// TIA Portal V16 export
// export: Created 2024-12-03T15:41:41.7978577Z, ExportSetting WithDefaults, DisplayName Totally Integrated Automation Portal, DisplayVersion V16 Update 6, DisplayName TIA Portal Version Control Interface, DisplayVersion V16 Update 2, DisplayName TIA Portal Openness, DisplayVersion V16 Update 6, DisplayName TIA Portal Teamcenter Gateway, DisplayVersion V16, DisplayName SINAMICS Startdrive Advanced, DisplayVersion V16 Update 5, DisplayName SINAMICS Startdrive G130, G150, S120, S150, SINAMICS MV, S210, DisplayVersion V16 Update 5, DisplayName SINAMICS Startdrive G110M, G120, G120C, G120D, G120P, G115D, DisplayVersion V16 Update 5, DisplayName STEP 7 Professional, DisplayVersion V16 Update 6, DisplayName STEP 7 Safety, DisplayVersion V16, DisplayName WinCC Advanced / Unified PC, DisplayVersion V16 Update 6
FUNCTION_BLOCK "EasySystems_TransferUnit_UpDown_Controller_FB"   // FB33, SCL
{ S7_Optimized_Access := 'TRUE' }
VERSION : 0.1
// stored: AutoNumber true, IsIECCheckEnabled false, IsRetainMemResEnabled false, MemoryReserve 100, SetENOAutomatically false, UDAEnableTagReadback false
   VAR_INPUT
      I_MotorData : "CLXAiPLC_IN_UDT";   // The 64 byte input word of the IO module
      I_ControlLeftMotorConveyLInx : Bool;   // 1 = control left motor both motos can be controlled with one module
      I_ControlRightMotorConveyLinx : Bool;   // 1 = control right motor both motors can be controlled with one fb
      I_UpFb : Bool;   // Object is up feedback
      I_DownFb : Bool;   // Object is down feedback
      I_TimeUp : Time := t#5s;   // time to go up
      I_TimeDown : Time := t#5s;   // time to go down
      I_Direction : Bool;   // Direction of the motor
   END_VAR
   VAR_IN_OUT
      IO_MotorStatus : "EasySystems_LineairMotor_ConveyLinx_FullPLC_Single";
      IO_MotorOutput : "CLXAiPLC_OUT_UDT";   // All the motor commands
   END_VAR
   VAR
      SensorUp : "SmartBool";
      SensorDown : "SmartBool";
      NotConnected { S7_SetPoint := 'True'} : TON_TIME;
      NotUp { S7_SetPoint := 'True'} : TON_TIME;
      NotDown { S7_SetPoint := 'True'} : TON_TIME;
      srUp { S7_SetPoint := 'True'} : "SR";
      srDown { S7_SetPoint := 'True'} : "SR";
      CycleRun { S7_SetPoint := 'True'} : "CycleRun";
   END_VAR
   VAR DB_SPECIFIC
      AlarmInfo { S7_SetPoint := 'True'} : "AlarmInfo_UDT";
   END_VAR
   VAR
      Overheat { S7_SetPoint := 'True'} : Program_Alarm;
      ShortCircuit { S7_SetPoint := 'True'} : Program_Alarm;
      MDRNotConnected { S7_SetPoint := 'True'} : Program_Alarm;
      Overload { S7_SetPoint := 'True'} : Program_Alarm;
      Stalled { S7_SetPoint := 'True'} : Program_Alarm;
      MDRBadHall { S7_SetPoint := 'True'} : Program_Alarm;
      OverVoltage { S7_SetPoint := 'True'} : Program_Alarm;
      LowVoltage { S7_SetPoint := 'True'} : Program_Alarm;
      NotConnectedAlarm { S7_SetPoint := 'True'} : Program_Alarm;
      ConnectionNotOK { S7_SetPoint := 'True'} : Program_Alarm;
      AnyErrorActive { S7_SetPoint := 'True'} : Program_Alarm;
      JamError { S7_SetPoint := 'True'} : Program_Alarm;
      SensorLowGain { S7_SetPoint := 'True'} : Program_Alarm;
      NotUpAlarm { S7_SetPoint := 'True'} : Program_Alarm;
      NotDownAlarm { S7_SetPoint := 'True'} : Program_Alarm;
   END_VAR
   VAR_TEMP
      T_RunAuto : Bool;
      T_RunManual : Bool;
      T_AppState : "ApplicationState_UDT";
      T_ZoneInfo : "ZoneInfo";
   END_VAR
BEGIN
   #T_ZoneInfo := "ApplicationState_DB".ZoneNames[#IO_MotorStatus.Zone];
   #T_AppState := "ApplicationState_DB".Appstate[#T_ZoneInfo.AppStateIndex];
   #CycleRun(I_End:=15);

   REGION SENSOR INTERFACING

       #SensorUp(I_Sensor:=#I_UpFb);
       #SensorDown(I_Sensor := #I_DownFb);

   END_REGION

   REGION Commands

       //Transfer unit settings
       #IO_MotorStatus.Cmd.Accel := 80;
       #IO_MotorStatus.Cmd.Deaccel := 1;
       #IO_MotorStatus.Cmd.SpeedManual := 20;
       #IO_MotorStatus.Cmd.SpeedAuto := 20;
       #IO_MotorStatus.Cmd.BrakeMode := 16#3;

       #IO_MotorStatus.Status.ManualCommandsDisabled := 0;

       //Reset commands left
       IF #I_ControlLeftMotorConveyLInx THEN
           #IO_MotorOutput.LeftMDRControl.MDR_Direction := 0;
           #IO_MotorOutput.LeftMDRControl.Run_MDR := 0;
           #IO_MotorOutput.LeftMDRSpeed := 0;
           #IO_MotorOutput.ServoControlCommandLeft.ResetPulseCount := 0;
           #IO_MotorOutput.ServoControlCommandLeft.RunToSetpoint := 0;
           #IO_MotorOutput.LeftMDRAccel := #IO_MotorStatus.Cmd.Accel;
           #IO_MotorOutput.LeftMDRDeccel := #IO_MotorStatus.Cmd.Deaccel;
           #IO_MotorOutput.LeftMDRBrakeMode := #IO_MotorStatus.Cmd.BrakeMode;
       END_IF;

       //Reset commands right
       IF #I_ControlRightMotorConveyLinx THEN
           #IO_MotorOutput.RightMDRControl.MDR_Direction := 0;
           #IO_MotorOutput.RightMDRControl.Run_MDR := 0;
           #IO_MotorOutput.RightMDRSpeed := 0;
           #IO_MotorOutput.ServoControlCommandRight.ResetPulseCount := 0;
           #IO_MotorOutput.ServoControlCommandRight.RunToSetpoint := 0;
           #IO_MotorOutput.RightMDRAccel := #IO_MotorStatus.Cmd.Accel;
           #IO_MotorOutput.RightMDRDeccel := #IO_MotorStatus.Cmd.Deaccel;
           #IO_MotorOutput.RightMDRBrakeMode := #IO_MotorStatus.Cmd.BrakeMode;
       END_IF;

       //INIT command
       IF #IO_MotorStatus.Cmd.InitPosition THEN
           #IO_MotorStatus.Status.PositionLineair := 0;
           #IO_MotorStatus.Cmd.InitPosition := FALSE;
       END_IF;

       IF #IO_MotorStatus.Status.PositionLineair = 1 THEN
           #IO_MotorStatus.Cmd.UpManual := 0;
           #IO_MotorStatus.Cmd.UpAuto := 0;
       END_IF;

       IF #IO_MotorStatus.Status.PositionLineair = -1 THEN
           #IO_MotorStatus.Cmd.DownAuto := 0;
           #IO_MotorStatus.Cmd.DownManual := 0;
       END_IF;

       IF #SensorUp.O_data.LE OR #SensorDown.O_data.LE THEN
           #IO_MotorStatus.Status.ManualCommandsDisabled := 1;
       END_IF;

       #T_RunAuto := #IO_MotorStatus.Cmd.UpAuto OR #IO_MotorStatus.Cmd.DownAuto;
       #T_RunManual := #IO_MotorStatus.Cmd.UpManual OR #IO_MotorStatus.Cmd.DownManual;

       //Turn commands of if manual mode is deactivated
       IF NOT #T_AppState.States.ManualModeActivated.State THEN
           #IO_MotorStatus.Cmd.UpManual := 0;
           #IO_MotorStatus.Cmd.DownManual := 0;
           #T_RunManual := 0;
           #IO_MotorStatus.Status.ManualCommandsDisabled := 1;
       END_IF;

       //Turn commands of if auto mode is deactivated
       IF NOT #T_AppState.States.AutoModeActivated.State THEN
           #IO_MotorStatus.Cmd.UpAuto := 0;
           #IO_MotorStatus.Cmd.DownAuto := 0;
           #T_RunAuto := 0;
       END_IF;

       //Turn commands of if interlock or alarm
       IF #IO_MotorStatus.Alarms.Status > 0 OR #IO_MotorStatus.Alarms.MdrAlarms.Status_1 > 0 OR #IO_MotorStatus.Status.Interlocked THEN
           #T_RunAuto := 0;
           #T_RunManual := 0;
           #IO_MotorStatus.Cmd.DownAuto := 0;
           #IO_MotorStatus.Cmd.DownManual := 0;
           #IO_MotorStatus.Cmd.UpAuto := 0;
           #IO_MotorStatus.Cmd.UpManual := 0;
           #IO_MotorStatus.Status.ManualCommandsDisabled := 1;
       END_IF;

       //Auto mode left
       IF #T_AppState.States.AutoModeActivated.State AND #I_ControlLeftMotorConveyLInx THEN
           #IO_MotorOutput.LeftMDRControl.Run_MDR := #T_RunAuto;
           #IO_MotorOutput.LeftMDRControl.MDR_Direction := #I_Direction;
           #IO_MotorOutput.LeftMDRAccel := #IO_MotorStatus.Cmd.Accel;
           #IO_MotorOutput.LeftMDRDeccel := #IO_MotorStatus.Cmd.Deaccel;
           #IO_MotorOutput.LeftMDRSpeed := #IO_MotorStatus.Cmd.SpeedAuto;
           #IO_MotorOutput.LeftMDRBrakeMode := #IO_MotorStatus.Cmd.BrakeMode;
           #IO_MotorOutput.ServoControlCommandLeft.ResetPulseCount := #IO_MotorStatus.Cmd.ServoResetPulseCount;
           #IO_MotorOutput.ServoControlCommandLeft.RunToSetpoint := #IO_MotorStatus.Cmd.ServoRunToSetpoint;
           #IO_MotorOutput.ServoControlDistanceLeft := #IO_MotorStatus.Cmd.ServoControlDistance;
       END_IF;

       //Auto mode right
       IF #T_AppState.States.AutoModeActivated.State AND #I_ControlRightMotorConveyLinx THEN
           #IO_MotorOutput.RightMDRControl.Run_MDR := #T_RunAuto;
           #IO_MotorOutput.RightMDRControl.MDR_Direction := #I_Direction;
           #IO_MotorOutput.RightMDRAccel := #IO_MotorStatus.Cmd.Accel;
           #IO_MotorOutput.RightMDRDeccel := #IO_MotorStatus.Cmd.Deaccel;
           #IO_MotorOutput.RightMDRSpeed := #IO_MotorStatus.Cmd.SpeedAuto;
           #IO_MotorOutput.RightMDRBrakeMode := #IO_MotorStatus.Cmd.BrakeMode;
           #IO_MotorOutput.ServoControlCommandRight.ResetPulseCount := #IO_MotorStatus.Cmd.ServoResetPulseCount;
           #IO_MotorOutput.ServoControlCommandRight.RunToSetpoint := #IO_MotorStatus.Cmd.ServoRunToSetpoint;
           #IO_MotorOutput.ServoControlDistanceRight := #IO_MotorStatus.Cmd.ServoControlDistance;
       END_IF;

       //Manual mode left
       IF #T_AppState.States.ManualModeActivated.State AND #I_ControlLeftMotorConveyLInx THEN
           #IO_MotorOutput.LeftMDRControl.MDR_Direction := #I_Direction;
           #IO_MotorOutput.LeftMDRControl.Run_MDR := #T_RunManual;
           #IO_MotorOutput.LeftMDRSpeed := #IO_MotorStatus.Cmd.SpeedManual;
       END_IF;

       //Manual mode right
       IF #T_AppState.States.ManualModeActivated.State AND #I_ControlRightMotorConveyLinx THEN
           #IO_MotorOutput.RightMDRControl.MDR_Direction := #I_Direction;
           #IO_MotorOutput.RightMDRControl.Run_MDR := #T_RunManual;
           #IO_MotorOutput.RightMDRSpeed := #IO_MotorStatus.Cmd.SpeedManual;
       END_IF;

       //Default commands
       IF  #I_ControlLeftMotorConveyLInx THEN
           #IO_MotorOutput.LeftMDRAccel := #IO_MotorStatus.Cmd.Accel := 30;
           #IO_MotorOutput.LeftMDRDeccel := #IO_MotorStatus.Cmd.Deaccel := 1;
           #IO_MotorOutput.LeftMDRSpeed := #IO_MotorStatus.Cmd.SpeedAuto := 50;
           #IO_MotorOutput.LeftMDRBrakeMode := #IO_MotorStatus.Cmd.BrakeMode;
       END_IF;

       IF #I_ControlRightMotorConveyLinx THEN
           #IO_MotorOutput.RightMDRAccel := #IO_MotorStatus.Cmd.Accel;
           #IO_MotorOutput.RightMDRDeccel := #IO_MotorStatus.Cmd.Deaccel;
           #IO_MotorOutput.RightMDRSpeed := #IO_MotorStatus.Cmd.SpeedAuto;
           #IO_MotorOutput.RightMDRBrakeMode := #IO_MotorStatus.Cmd.BrakeMode;
       END_IF;

   END_REGION

   REGION Interlock motor

       #IO_MotorStatus.Status.Interlocked := #IO_MotorStatus.Cmd.Interlock OR NOT #T_AppState.States.EmergencyOk.State;
       #IO_MotorStatus.Status.Status.%X0 := #IO_MotorStatus.Status.Interlocked;

   END_REGION

   REGION Create status

       //Lineair position
       IF #SensorUp.O_data.State AND NOT #SensorDown.O_data.State THEN
           #IO_MotorStatus.Status.PositionLineair := 1;
       END_IF;

       IF NOT #SensorUp.O_data.State AND #SensorDown.O_data.State THEN
           #IO_MotorStatus.Status.PositionLineair := -1;
       END_IF;

       IF NOT #T_AppState.States.AutoModeActivated.State
           AND NOT #T_AppState.States.ManualModeActivated.State THEN
           #IO_MotorStatus.Status.PositionLineair := 0;
       END_IF;

       REGION simulation

           IF "Simulation_DB".Simulation_On THEN
               IF #IO_MotorStatus.Cmd.UpAuto OR #IO_MotorStatus.Cmd.UpManual THEN
                   #IO_MotorStatus.Status.PositionLineair := "Up";
               END_IF;
           END_IF;

           IF "Simulation_DB".Simulation_On THEN
               IF #IO_MotorStatus.Cmd.DownAuto OR #IO_MotorStatus.Cmd.DownManual THEN
                   #IO_MotorStatus.Status.PositionLineair := "Down";
               END_IF;
           END_IF;

       END_REGION

       //Left
       IF #I_ControlLeftMotorConveyLInx THEN
           #IO_MotorStatus.Status.ActualSpeed := #I_MotorData.LeftMDRRealSpeed;
           #IO_MotorStatus.Status.Current := #I_MotorData.LeftCurrent;
           #IO_MotorStatus.Status.Frequency := #I_MotorData.LeftFreq;
           #IO_MotorStatus.Status.ManualModeActive := #IO_MotorStatus.Cmd.UpManual OR #IO_MotorStatus.Cmd.DownManual;
           #IO_MotorStatus.Status.Position := #I_MotorData.DistanceLeft;
           #IO_MotorStatus.Status.Running := #I_MotorData.LeftMDRRealSpeed > 0 AND #IO_MotorOutput.LeftMDRControl.Run_MDR;
           #IO_MotorStatus.Status.ServoStatus.LastServoCommandExecuted := #I_MotorData.ServoStatusLeft.LastServoCommandExecuted;
           #IO_MotorStatus.Status.ServoStatus.ResetPulseCount_Echo := #I_MotorData.ServoStatusLeft.ResetPulseCount_Echo;
           #IO_MotorStatus.Status.ServoStatus.RunCommand_Echo := #I_MotorData.ServoStatusLeft.RunCommand_Echo;
           #IO_MotorStatus.Status.TemperatureModule := #I_MotorData.ModuleTemp;
           #IO_MotorStatus.Status.TeperatureMDR := #I_MotorData.LeftCalcTemp;
       END_IF;

       //right
       IF #I_ControlRightMotorConveyLinx THEN
           #IO_MotorStatus.Status.ActualSpeed := #I_MotorData.RightMDRRealSpeed;
           #IO_MotorStatus.Status.Current := #I_MotorData.RightCurrent;
           #IO_MotorStatus.Status.Frequency := #I_MotorData.RightFreq;
           #IO_MotorStatus.Status.ManualModeActive := #IO_MotorStatus.Cmd.UpManual OR #IO_MotorStatus.Cmd.DownManual;
           #IO_MotorStatus.Status.Position := #I_MotorData.DistanceRight;
           #IO_MotorStatus.Status.Running := #I_MotorData.RightMDRRealSpeed > 0 AND #IO_MotorOutput.RightMDRControl.Run_MDR;
           #IO_MotorStatus.Status.ServoStatus.LastServoCommandExecuted := #I_MotorData.ServoStatusRight.LastServoCommandExecuted;
           #IO_MotorStatus.Status.ServoStatus.ResetPulseCount_Echo := #I_MotorData.ServoStatusRight.ResetPulseCount_Echo;
           #IO_MotorStatus.Status.ServoStatus.RunCommand_Echo := #I_MotorData.ServoStatusRight.RunCommand_Echo;
           #IO_MotorStatus.Status.TemperatureModule := #I_MotorData.ModuleTemp;
           #IO_MotorStatus.Status.TeperatureMDR := #I_MotorData.RightCalcTemp;
       END_IF;

       REGION Min max voltage

           #IO_MotorStatus.Status.Voltage := #I_MotorData.Voltage;
           IF #I_MotorData.Voltage < #IO_MotorStatus.Status.MinVoltage THEN
               #IO_MotorStatus.Status.MinVoltage := #I_MotorData.Voltage;
           END_IF;

           IF #I_MotorData.Voltage > #IO_MotorStatus.Status.MaxVoltage THEN
               #IO_MotorStatus.Status.MaxVoltage := #I_MotorData.Voltage;
           END_IF;

       END_REGION

       #IO_MotorStatus.Status.ManualModeActive := #T_AppState.States.ManualModeActivated.State;
       #IO_MotorStatus.Status.Status.%X1 := #IO_MotorStatus.Status.Running;
       #IO_MotorStatus.Status.Status.%X2 := #IO_MotorStatus.Status.ManualModeActive;

   END_REGION

   REGION Check alarm active

       IF #I_ControlLeftMotorConveyLInx THEN

           IF #I_MotorData.LeftMDRDiagnostic.LowVoltage THEN
               #IO_MotorStatus.Alarms.MdrAlarms.LowVoltage.Active := True;
           END_IF;

           IF #I_MotorData.LeftMDRDiagnostic.MDRBadHall THEN
               #IO_MotorStatus.Alarms.MdrAlarms.MDRBadHall.Active := True;
           END_IF;

           IF #I_MotorData.LeftMDRDiagnostic.MDRNotConnected THEN
               #IO_MotorStatus.Alarms.MdrAlarms.MDRNotConnected.Active := True;
           END_IF;

           IF #I_MotorData.LeftMDRDiagnostic.Overheat THEN
               #IO_MotorStatus.Alarms.MdrAlarms.Overheat.Active := True;
           END_IF;

           IF #I_MotorData.LeftMDRDiagnostic.Overload THEN
               #IO_MotorStatus.Alarms.MdrAlarms.Overload.Active := True;
           END_IF;

           IF #I_MotorData.LeftMDRDiagnostic.OverVoltage THEN
               #IO_MotorStatus.Alarms.MdrAlarms.OverVoltage.Active := True;
           END_IF;

           IF #I_MotorData.LeftMDRDiagnostic.ShortCircuit THEN
               #IO_MotorStatus.Alarms.MdrAlarms.ShortCircuit.Active := True;
           END_IF;

           IF #I_MotorData.LeftMDRDiagnostic.Stalled THEN
               #IO_MotorStatus.Alarms.MdrAlarms.Stalled.Active := True;
           END_IF;

       END_IF;

       IF #I_ControlRightMotorConveyLinx THEN

           IF #I_MotorData.RightMDRDiagnostic.LowVoltage THEN
               #IO_MotorStatus.Alarms.MdrAlarms.LowVoltage.Active := True;
           END_IF;

           IF #I_MotorData.RightMDRDiagnostic.MDRBadHall THEN
               #IO_MotorStatus.Alarms.MdrAlarms.MDRBadHall.Active := True;
           END_IF;

           IF #I_MotorData.RightMDRDiagnostic.MDRNotConnected THEN
               #IO_MotorStatus.Alarms.MdrAlarms.MDRNotConnected.Active := True;
           END_IF;

           IF #I_MotorData.RightMDRDiagnostic.Overheat THEN
               #IO_MotorStatus.Alarms.MdrAlarms.Overheat.Active := True;
           END_IF;

           IF #I_MotorData.RightMDRDiagnostic.Overload THEN
               #IO_MotorStatus.Alarms.MdrAlarms.Overload.Active := True;
           END_IF;

           IF #I_MotorData.RightMDRDiagnostic.OverVoltage THEN
               #IO_MotorStatus.Alarms.MdrAlarms.OverVoltage.Active := True;
           END_IF;

           IF #I_MotorData.RightMDRDiagnostic.ShortCircuit THEN
               #IO_MotorStatus.Alarms.MdrAlarms.ShortCircuit.Active := True;
           END_IF;

           IF #I_MotorData.RightMDRDiagnostic.Stalled THEN
               #IO_MotorStatus.Alarms.MdrAlarms.Stalled.Active := True;
           END_IF;

       END_IF;

       #IO_MotorStatus.Heartbeat := #I_MotorData.AllSensors.Heartbeat;
       #NotConnected(IN := NOT #IO_MotorStatus.Heartbeat,
                       PT := t#5s);

       IF #NotConnected.Q THEN
           #IO_MotorStatus.Alarms.MdrAlarms.NotConnected.Active := true;
       END_IF;

       //Not up
       #NotUp(IN := (#IO_MotorStatus.Cmd.UpAuto OR #IO_MotorStatus.Cmd.UpManual) AND NOT #SensorUp.O_data.State,
                PT := #I_TimeUp);

       #srUp(I_set := #NotUp.Q,
               I_Reset := #T_AppState.Hmi_Buttons.reset.state.State,
               O_state => #IO_MotorStatus.Alarms.NotUp.Active);

       //Not down
         #NotDown(IN := (#IO_MotorStatus.Cmd.DownAuto OR #IO_MotorStatus.Cmd.DownManual) AND NOT #SensorDown.O_data.State,
                  PT := #I_TimeDown);

       #srDown(I_set := #NotDown.Q,
                 I_Reset := #T_AppState.Hmi_Buttons.reset.state.State,
                 O_state => #IO_MotorStatus.Alarms.NotDown.Active);

       REGION PROGRAM ALARMS

           REGION alarm info
               IF NOT #AlarmInfo.init THEN
                   #IO_MotorStatus.Info.Name := "buildObjectName"(I_Symbolname := GetSymbolName(variable := #IO_MotorStatus,size := 100));
                   #AlarmInfo.info := "buildAlarmInfo"(I_ZoneIndex := #IO_MotorStatus.Zone, I_ZoneName := #T_ZoneInfo.ZoneName, I_ObjectName := #IO_MotorStatus.Info.Name);
                   #AlarmInfo.init := TRUE;
               END_IF;
           END_REGION

           REGION PROGRAM ALARMS MDR

               IF #CycleRun.O_Cycle = 1 THEN
                   #Overheat(SIG := #IO_MotorStatus.Alarms.MdrAlarms.Overheat.Active,
                             SD_1 := #T_ZoneInfo.ZoneName,
                             SD_2 := #IO_MotorStatus.Info.Name,
                             SD_3 := #AlarmInfo.info);
               END_IF;

               IF #CycleRun.O_Cycle = 2 THEN
                   #ShortCircuit(SIG := #IO_MotorStatus.Alarms.MdrAlarms.ShortCircuit.Active,
                                 SD_1 := #T_ZoneInfo.ZoneName,
                                 SD_2 := #IO_MotorStatus.Info.Name,
                                 SD_3 := #AlarmInfo.info);
               END_IF;

               IF #CycleRun.O_Cycle = 3 THEN
                   #MDRNotConnected(SIG := #IO_MotorStatus.Alarms.MdrAlarms.MDRNotConnected.Active,
                                    SD_1 := #T_ZoneInfo.ZoneName,
                                    SD_2 := #IO_MotorStatus.Info.Name,
                                    SD_3 := #AlarmInfo.info);
               END_IF;

               IF #CycleRun.O_Cycle = 4 THEN
                   #Overload(SIG := #IO_MotorStatus.Alarms.MdrAlarms.Overload.Active,
                             SD_1 := #T_ZoneInfo.ZoneName,
                             SD_2 := #IO_MotorStatus.Info.Name,
                             SD_3 := #AlarmInfo.info);
               END_IF;

               IF #CycleRun.O_Cycle = 5 THEN
                   #Stalled(SIG := #IO_MotorStatus.Alarms.MdrAlarms.Stalled.Active,
                            SD_1 := #T_ZoneInfo.ZoneName,
                            SD_2 := #IO_MotorStatus.Info.Name,
                            SD_3 := #AlarmInfo.info);
               END_IF;

               IF #CycleRun.O_Cycle = 6 THEN
                   #MDRBadHall(SIG := #IO_MotorStatus.Alarms.MdrAlarms.MDRBadHall.Active,
                               SD_1 := #T_ZoneInfo.ZoneName,
                               SD_2 := #IO_MotorStatus.Info.Name,
                               SD_3 := #AlarmInfo.info);
               END_IF;

                   IF #CycleRun.O_Cycle = 7 THEN
                       #OverVoltage(SIG := #IO_MotorStatus.Alarms.MdrAlarms.OverVoltage.Active,
                                    SD_1 := #T_ZoneInfo.ZoneName,
                                    SD_2 := #IO_MotorStatus.Info.Name,
                                    SD_3 := #AlarmInfo.info);
                   END_IF;

                   IF #CycleRun.O_Cycle = 8 THEN
                       #LowVoltage(SIG := #IO_MotorStatus.Alarms.MdrAlarms.LowVoltage.Active,
                                   SD_1 := #T_ZoneInfo.ZoneName,
                                   SD_2 := #IO_MotorStatus.Info.Name,
                                   SD_3 := #AlarmInfo.info);
                   END_IF;

                   IF #CycleRun.O_Cycle = 9 THEN
                       #NotConnectedAlarm(SIG := #IO_MotorStatus.Alarms.MdrAlarms.NotConnected.Active,
                                     SD_1 := #T_ZoneInfo.ZoneName,
                                     SD_2 := #IO_MotorStatus.Info.Name,
                                     SD_3 := #AlarmInfo.info);
                   END_IF;

                   IF #CycleRun.O_Cycle = 10 THEN
                       #ConnectionNotOK(SIG := #IO_MotorStatus.Alarms.MdrAlarms.ConnectionNotOK.Active,
                                        SD_1 := #T_ZoneInfo.ZoneName,
                                        SD_2 := #IO_MotorStatus.Info.Name,
                                        SD_3 := #AlarmInfo.info);
                   END_IF;

                   IF #CycleRun.O_Cycle = 11 THEN
                       #AnyErrorActive(SIG := #IO_MotorStatus.Alarms.MdrAlarms.AnyErrorActive.Active,
                                       SD_1 := #T_ZoneInfo.ZoneName,
                                       SD_2 := #IO_MotorStatus.Info.Name,
                                       SD_3 := #AlarmInfo.info);
                   END_IF;

                   IF #CycleRun.O_Cycle = 12 THEN
                       #JamError(SIG := #IO_MotorStatus.Alarms.MdrAlarms.JamError.Active,
                                 SD_1 := #T_ZoneInfo.ZoneName,
                                 SD_2 := #IO_MotorStatus.Info.Name,
                                 SD_3 := #AlarmInfo.info);
                   END_IF;

                   IF #CycleRun.O_Cycle = 13 THEN
                       #SensorLowGain(SIG := #IO_MotorStatus.Alarms.MdrAlarms.SensorLowGain.Active,
                                      SD_1 := #T_ZoneInfo.ZoneName,
                                      SD_2 := #IO_MotorStatus.Info.Name,
                                      SD_3 := #AlarmInfo.info);
                   END_IF;

           END_REGION

           REGION PROGRAM ALARMS TRANSFER UNIT

               IF #CycleRun.O_Cycle = 14 THEN
                   #NotUpAlarm(SIG := #IO_MotorStatus.Alarms.NotUp.Active,
                          SD_1 := #T_ZoneInfo.ZoneName,
                          SD_2 := #IO_MotorStatus.Info.Name,
                          SD_3 := #AlarmInfo.info);
               END_IF;

               IF #CycleRun.O_Cycle = 15 THEN
                   #NotDownAlarm(SIG := #IO_MotorStatus.Alarms.NotDown.Active,
                            SD_1 := #T_ZoneInfo.ZoneName,
                            SD_2 := #IO_MotorStatus.Info.Name,
                            SD_3 := #AlarmInfo.info);
               END_IF;


           END_REGION

       END_REGION

   END_REGION

   REGION Alarm status

       #IO_MotorStatus.Alarms.Status.%X0 := #IO_MotorStatus.Alarms.NotUp.Active;
       #IO_MotorStatus.Alarms.Status.%X1 := #IO_MotorStatus.Alarms.NotDown.Active;
       #IO_MotorStatus.Alarms.Status.%X2 := #IO_MotorStatus.Alarms.MdrAlarms.Status_1 > 0;

       REGION MDR alarms

           #IO_MotorStatus.Alarms.MdrAlarms.Status_1.%X0 := #IO_MotorStatus.Alarms.MdrAlarms.Overheat.Active;
           //#MotorStatus.Alarms.MdrAlarms.Status_1.%X1 := #MotorStatus.Alarms.MdrAlarms.Overheat.Active;
           #IO_MotorStatus.Alarms.MdrAlarms.Status_1.%X2 := #IO_MotorStatus.Alarms.MdrAlarms.ShortCircuit.Active;
           #IO_MotorStatus.Alarms.MdrAlarms.Status_1.%X3 := #IO_MotorStatus.Alarms.MdrAlarms.MDRNotConnected.Active;

           #IO_MotorStatus.Alarms.MdrAlarms.Status_1.%X4 := #IO_MotorStatus.Alarms.MdrAlarms.Overload.Active;
           #IO_MotorStatus.Alarms.MdrAlarms.Status_1.%X5 := #IO_MotorStatus.Alarms.MdrAlarms.Stalled.Active;
           #IO_MotorStatus.Alarms.MdrAlarms.Status_1.%X6 := #IO_MotorStatus.Alarms.MdrAlarms.MDRBadHall.Active;
           // #MotorStatus.Alarms.MdrAlarms.Status_1.%X7 := #MotorStatus.Alarms.MdrAlarms.Overheat.Active;

           #IO_MotorStatus.Alarms.MdrAlarms.Status_1.%X8 := #IO_MotorStatus.Alarms.MdrAlarms.OverVoltage.Active;
           #IO_MotorStatus.Alarms.MdrAlarms.Status_1.%X9 := #IO_MotorStatus.Alarms.MdrAlarms.LowVoltage.Active;
           #IO_MotorStatus.Alarms.MdrAlarms.Status_1.%X10 := #IO_MotorStatus.Alarms.MdrAlarms.NotConnected.Active;
           #IO_MotorStatus.Alarms.MdrAlarms.Status_1.%X11 := #IO_MotorStatus.Alarms.MdrAlarms.ConnectionNotOK.Active;

           #IO_MotorStatus.Alarms.MdrAlarms.Status_1.%X12 := #IO_MotorStatus.Alarms.MdrAlarms.AnyErrorActive.Active;
           #IO_MotorStatus.Alarms.MdrAlarms.Status_1.%X13 := #IO_MotorStatus.Alarms.MdrAlarms.JamError.Active;
           #IO_MotorStatus.Alarms.MdrAlarms.Status_1.%X14 := #IO_MotorStatus.Alarms.MdrAlarms.SensorLowGain.Active;
           #IO_MotorStatus.Alarms.MdrAlarms.Status_1.%X15 := #IO_MotorStatus.Alarms.MdrAlarms.Overheat.Active;

       END_REGION

       IF #IO_MotorStatus.Alarms.Status > 0 THEN
           "ApplicationState_DB".Appstate[#T_ZoneInfo.AppStateIndex].Alarms.AlarmActiveInternalPLC := TRUE;
       END_IF;

   END_REGION

   REGION Reset alarms

       IF #IO_MotorStatus.Alarms.Status > 0 AND (#T_AppState.Hmi_Buttons.reset.state.State
           OR #IO_MotorStatus.Cmd.Reset
           OR "Simulation_DB".Simulation_On) THEN

           #IO_MotorStatus.Alarms.MdrAlarms.Overheat.Active := False;
           #IO_MotorStatus.Alarms.MdrAlarms.Overheat.Active := False;
           #IO_MotorStatus.Alarms.MdrAlarms.ShortCircuit.Active := False;
           #IO_MotorStatus.Alarms.MdrAlarms.MDRNotConnected.Active := False;

           #IO_MotorStatus.Alarms.MdrAlarms.Overload.Active := False;
           #IO_MotorStatus.Alarms.MdrAlarms.Stalled.Active := False;
           #IO_MotorStatus.Alarms.MdrAlarms.MDRBadHall.Active := False;
           #IO_MotorStatus.Alarms.MdrAlarms.Overheat.Active := False;
           #IO_MotorStatus.Alarms.MdrAlarms.OverVoltage.Active := False;
           #IO_MotorStatus.Alarms.MdrAlarms.LowVoltage.Active := False;
           #IO_MotorStatus.Alarms.MdrAlarms.NotConnected.Active := False;
           #IO_MotorStatus.Alarms.MdrAlarms.ConnectionNotOK.Active := False;

           #IO_MotorStatus.Alarms.MdrAlarms.AnyErrorActive.Active := False;
           #IO_MotorStatus.Alarms.MdrAlarms.JamError.Active := False;
           #IO_MotorStatus.Alarms.MdrAlarms.SensorLowGain.Active := False;
           #IO_MotorStatus.Alarms.MdrAlarms.Overheat.Active := False;

           #IO_MotorStatus.Alarms.NotDown.Active := 0;
           #IO_MotorStatus.Alarms.NotUp.Active := 0;

           #IO_MotorStatus.Alarms.Status := 0;
           #IO_MotorStatus.Alarms.MdrAlarms.Status_1 := 0;

       END_IF;

   END_REGION

   REGION common status
       #IO_MotorStatus.Info.CommonStatus := 0;
       IF #IO_MotorStatus.Status.Running THEN
           #IO_MotorStatus.Info.CommonStatus := 1;
       END_IF;

       IF #IO_MotorStatus.Alarms.Status > 1 THEN
           #IO_MotorStatus.Info.CommonStatus := -1;
       END_IF;
   END_REGION

   #IO_MotorStatus.Cmd.Reset := 0;
END_FUNCTION_BLOCK
